{attribute 'linkalways'} 
{attribute 'no_explicit_call' := 'This FB is a CLASS and must be accessed using methods or properties'}
{attribute 'enable_dynamic_creation'}
FUNCTION_BLOCK _DT EXTENDS DatatypeBase
VAR
	localData : DT;
	activeData : REFERENCE TO DT REF= localData;
END_VAR

PROPERTY PUBLIC Address : PVOID
GET
Address := ADR(activeData);
END_GET
END_PROPERTY

METHOD PUBLIC ClearReference
VAR_INPUT
END_VAR
activeData REF= localData;
END_METHOD

METHOD PUBLIC Clone : I_Datatype
VAR
    pClone : POINTER TO _DT;
END_VAR
pClone := __NEW(_DT(InitialValue := Value));
Clone := pClone^;
END_METHOD

METHOD FB_init : BOOL
VAR_INPUT
	bInitRetains : BOOL; // if TRUE, the retain variables are initialized (warm start / cold start)
	bInCopyCode : BOOL;  // if TRUE, the instance afterwards gets moved WORDo the copy code (online change)
	InitialValue : DT;
END_VAR
localData := InitialValue;
END_METHOD

METHOD PUBLIC MakeReferenceTo
VAR_INPUT
	ReferenceTarget : REFERENCE TO DT;
END_VAR
activeData REF= ReferenceTarget;
END_METHOD

METHOD PUBLIC SerializeWith
VAR_INPUT
	Serializer : I_Serializer;
END_VAR
Serializer.AddDateTime(activeData);
END_METHOD

PROPERTY PUBLIC Size : UDINT
GET
Size := SIZEOF(activeData);
END_GET
END_PROPERTY

METHOD TryDeserializeFrom : BOOL
VAR_INPUT
	Deserializer : I_Deserializer;
	Feedback : I_DeserializerFeedback;
END_VAR
TryDeserializeFrom := Deserializer.TryGetDateTime(activeData, Feedback);
END_METHOD

METHOD TryMakeReferenceTo : BOOL
VAR_INPUT
	Target : I_Datatype;
END_VAR
VAR
	pTargetData : POINTER TO DT;
END_VAR
IF NOT (Target.TypeName = TypeName) THEN
	RETURN;
END_IF

pTargetData := Target.Address;
activeData REF= pTargetData^;
TryMakeReferenceTo := TRUE;
END_METHOD

PROPERTY PUBLIC TypeName : T_MAXSTRING
GET
TypeName := 'DT';
END_GET
END_PROPERTY

PROPERTY PUBLIC Value : DT
GET
Value := activeData;
END_GET
SET
activeData := Value;
END_SET
END_PROPERTY

END_FUNCTION_BLOCK

(* stored: Version 1.1.0.1, ProductVersion 3.1.4024.12
   POU _DT: Id {177c2a9c-f4f0-070a-224e-ca78373654f5}, SpecialFunc None
   Folder Constructor: Id {5fae493d-5532-07f4-1a5c-0d684f523964}
   Property Address: Id {b5246887-e120-09f3-07ea-105f4140959b}
   Get Get: Id {d93473a5-5537-0512-18f6-b0bc69ead019}
   Method ClearReference: Id {388a0ac9-f03b-0845-29be-97258497e9b6}
   Method Clone: Id {67f7e7f7-0f49-0336-25c5-087aae0a7cf1}
   Method FB_init: Id {f9d4f26e-d621-0b3b-1bf6-76703c830692}
   Method MakeReferenceTo: Id {339bbf93-d92b-0211-37e1-06e1fd97ec68}
   Method SerializeWith: Id {2dfca9e8-9c63-0315-17c1-6e898814597d}
   Property Size: Id {fd603935-c7b0-04c3-20ed-2cd623cc51bf}
   Get Get: Id {2c676d8b-4927-0919-3ac2-b005df33d289}
   Method TryDeserializeFrom: Id {054d3601-12ee-077a-2fa0-3d34ed70bf4d}
   Method TryMakeReferenceTo: Id {3038c7a9-cdba-03e8-34da-8365ae4db83f}
   Property TypeName: Id {f4b1d5b4-9629-0c80-2c73-86402d4ee55c}
   Get Get: Id {edadc259-0c52-08f7-1083-0037a59b80bc}
   Property Value: Id {73c5b951-8017-048f-2510-7fdb1fe52c8e}
   Get Get: Id {36acd71a-ccf2-0377-009c-cfdf5a4b70b7}
   Set Set: Id {00fc4b97-2496-0328-06b6-d05323815bb6} *)
